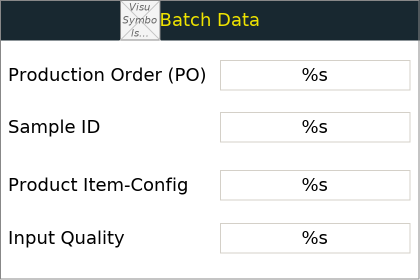
VISUALIZATION AOIBatchDataFrame  // 420x280
VAR_IN_OUT
	stBatchDataFrame : ST_BatchData;
END_VAR
    Label (5,170 210x30), "Product Item-Config"
    Label (5,223 210x30), "Input Quality"
    Textfield (220,170 190x30), "%s", text variable: stBatchDataFrame.sProductItemConfig
    Textfield (220,223 190x30), "%s", text variable: stBatchDataFrame.sInputQuantity
    Rectangle (0,0 420x40), "Batch Data"
    Image (120,0 40x40), image: VisuSymbols.Symbols.Database2
    Label (5,60 210x30), "Production Order (PO)"
    Label (5,112 210x30), "Sample ID"
    Textfield (220,60 190x30), "%s", text variable: stBatchDataFrame.sProductionOrder
    Textfield (220,112 190x30), "%s", text variable: stBatchDataFrame.sTrayID
END_VISUALIZATION

(* stored: Version 1.1.0.1, ProductVersion 3.1.4024.9
   Visu AOIBatchDataFrame: Id {50a70a8a-3065-4c5c-b551-db5804e770bc} *)
